FUNCTION_BLOCK UNSCALE (* Converts scaled UINT input of 0-100% to a D/A output value *)
  (* Standard: 61499-1 *)
  (* Version 0.0, 2004-09-01, JHC, Rockwell Automation *)
  (* Compiler header: package fb.rt.process; *)
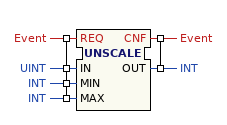
  EVENT_INPUT
    REQ WITH IN, MIN, MAX; (* Normal Execution Request *)
  END_EVENT
  EVENT_OUTPUT
    CNF WITH OUT; (* Execution Confirmation *)
  END_EVENT
  VAR_INPUT
    IN : UINT; (* Scaled Input, 0-100% *)
    MIN : INT; (* OUT value corresponding to IN=0 *)
    MAX : INT; (* OUT value corresponding to IN=100%, e.g., 4096 for a 12-bit D/A *)
  END_VAR
  VAR_OUTPUT
    OUT : INT; (* D/A Output corresponding to IN value, limited to {MIN..MAX-1} *)
  END_VAR
END_FUNCTION_BLOCK
